// Mitsubishi GX Works2 project: 6   PLC: FX2N/FX2NC

PROGRAM MAIN
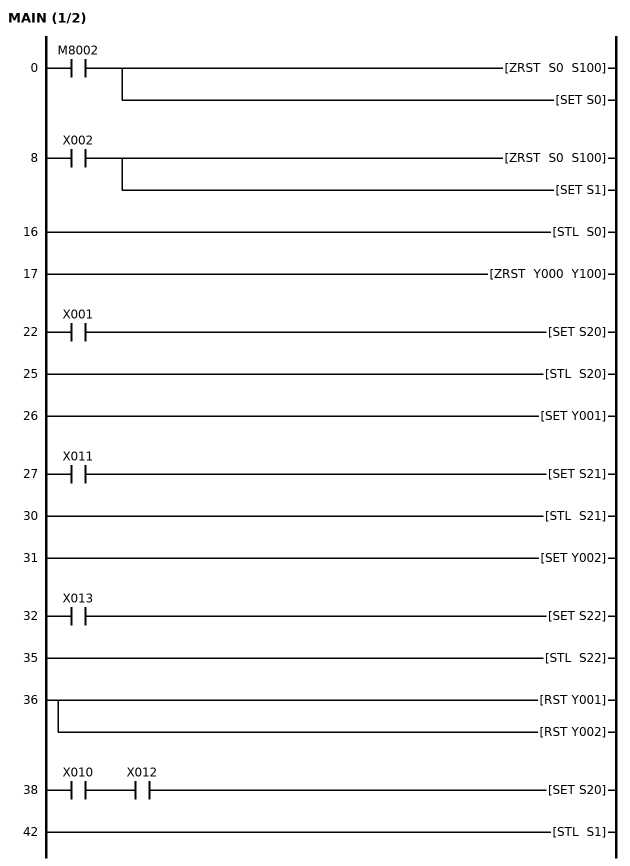
0     LD      M8002
      ZRST    S0 S100
      SET     S0
8     LD      X002
      ZRST    S0 S100
      SET     S1
16    STL     S0
17    ZRST    Y000 Y100
22    LD      X001
      SET     S20
25    STL     S20
26    SET     Y001
27    LD      X011
      SET     S21
30    STL     S21
31    SET     Y002
32    LD      X013
      SET     S22
35    STL     S22
36    RST     Y001
      RST     Y002
38    LD      X010
      AND     X012
      SET     S20
42    STL     S1
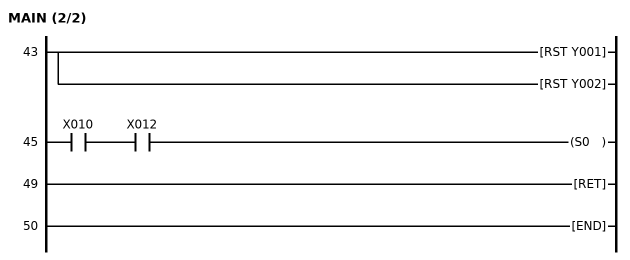
43    RST     Y001
      RST     Y002
45    LD      X010
      AND     X012
      OUT     S0
49    RET
50    END
END_PROGRAM

// device comments not shown above
BL0  ; main
BL1  ; a
BL2  ; b
